# B&R Automation Studio project AS_lab_4
Automation Studio 4.5.2.102

## Configuration Real

### Task classes (Cpu.sw)
```
Cyclic#1 (cycle 2000 us, tolerance 0 us):
  SDCAxisCtr <- SDCAxisCtrlX.prg
  SDCAxisCt1 <- SDCAxisCtrlY.prg
  SDCAxisCt2 <- SDCAxisCtrlZ.prg
DataObjects: Acp10sys
NcDataObjects: acp10etxen <- acp10etxen.dob, Axis_Xa <- AxisParameters.Axis_Xobj.Axis_Xa.dob, Axis_Xi <- AxisParameters.Axis_Xobj.Axis_Xi.dob, gmcipvar <- GmcIpUserConfig.gmcipvar.dob, gmcipfun <- GmcIpUserConfig.gmcipfun.dob, gmcipfub <- GmcIpUserConfig.gmcipfub.dob, gmcipubr <- GmcIpUserConfig.gmcipubr.dob, gmcipusm <- GmcIpUserConfig.gmcipusm.dob, gmcipui <- GmcIpUserConfig.gmcipui.dob, gmcipus <- GmcIpUserConfig.gmcipus.dob, gmcipuc <- GmcIpUserConfig.gmcipuc.dob, gmcipsys <- GmcIpConfig.gmcipsys.dob, gmciplbr <- GmcIpConfig.gmciplbr.dob, gmcipcbr <- GmcIpConfig.gmcipcbr.dob, gmciplsm <- GmcIpConfig.gmciplsm.dob, gmcipcsm <- GmcIpConfig.gmcipcsm.dob, gmcipcfg <- GmcIpConfig.gmcipcfg.dob, gmcipiec <- GmcIpConfig.gmcipiec.dob, gmciplog <- GmcIpConfig.gmciplog.dob, gmcipesm <- GmcIpConfig.gmcipesm.dob, gmcipmxd <- GmcIpConfig.gmcipmxd.dob, gmcipmx <- GmcIpConfig.gmcipmx.dob, CncInit <- CNC.CncInit.dob, CncProg <- CNC.CncProg.dob
VcDataObjects: GUI <- GUI.dob
Binaries: TCData, udbdef, vcpdsw, vcrt, vcmgr, vcctext, vcpfmtcx, vccslider, vcfile, vcgclass, arial, vcdsint, vcdsloc, vcfntttf, GUI01, GUI03, GUI02, vccovl, vcshared, arialbd, vcalarm, vcptelo, vccdt, vcpdpp30, vccbtn, vccnum, vcbclass, vcpfpp30, vctcal, ashwd, Role, User, sysconf, ashwac, asfw, arconfig, iomap, Acp10map, acp10cfg, Acp10map1
Libraries: Acp10man, Acp10par, NcGlobal, Acp10sdc, AsBrStr, Acp10_MC, brsystem, sys_lib, runtime, Acp10sim, AsIOTime, MotorCtrl, powerlnk, vcresman, Arnc0man, DataObj, AsArLog, FileIO, AsArProf, AsMem, astime
```

### Hardware
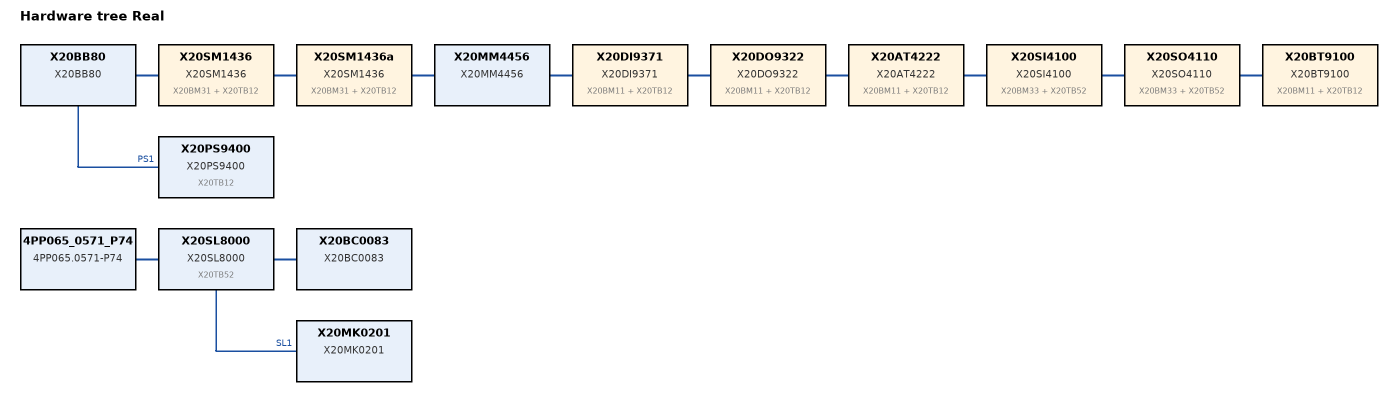
```
4PP065_0571_P74 : 4PP065.0571-P74 v1.1.2.0
  Connector IF5:
    ActivateDevice = 1
    Mode = Manual
    InternetAddress = 10.0.1.10
    SubnetMask = 255.255.255.0
  ConfigurationID = labBR
  Simulation = 1
  TimerDeviceType = EPLX2X
  TimerDevice = 4PP065_0571_P74.IF4
  TaskClassIdleTime = 2000
  Cyclic1Duration = 2000
  Cyclic1Tolerance = 0
  Cyclic1Output = 1
  Cyclic2Duration = 10000
  Cyclic2Tolerance = 10000
  VcObjectName = GUI
X20AT4222 : X20AT4222 v1.2.3.0  [SS1 -> X20TB12e.SS; SL -> X20BM11b.SL1]
X20BB80 : X20BB80 v1.0.2.0
X20BC0083 : X20BC0083 v2.8.0.0  [PLK1 -> X20SL8000.PLK2 [Cable Type=PowerlinkCable, Length=10, Version=1.0.0.2]; SL -> X20BB80.SL1]
X20BM11 : X20BM11 v1.0.0.1  [X2X1 -> X20MM4456.X2X2]
X20BM11a : X20BM11 v1.0.0.1  [X2X1 -> X20BM11.X2X2]
X20BM11b : X20BM11 v1.0.0.1  [X2X1 -> X20BM11a.X2X2]
X20BM11c : X20BM11 v1.0.0.1  [X2X1 -> X20BM33a.X2X2]
X20BM31 : X20BM31 v1.0.0.1  [X2X1 -> X20BB80.IF1]
X20BM31a : X20BM31 v1.0.0.1  [X2X1 -> X20BM31.X2X2]
X20BM33 : X20BM33 v1.0.0.4  [X2X1 -> X20BM11b.X2X2]
X20BM33a : X20BM33 v1.0.0.4  [X2X1 -> X20BM33.X2X2]
X20BT9100 : X20BT9100 v1.0.3.0  [SS1 -> X20TB12f.SS; SL -> X20BM11c.SL1]
X20DI9371 : X20DI9371 v1.0.2.0  [SS1 -> X20TB12c.SS; SL -> X20BM11.SL1]
X20DO9322 : X20DO9322 v1.0.3.0  [SS1 -> X20TB12d.SS; SL -> X20BM11a.SL1]
X20MK0201 : X20MK0201 v1.0.0.0  [SL -> X20SL8000.SL1]
X20MM4456 : X20MM4456 v1.1.5.0  [X2X1 -> X20BM31a.X2X2]
X20PS9400 : X20PS9400 v1.0.2.4  [SS1 -> X20TB12.SS; PS -> X20BB80.PS1]
X20SI4100 : X20SI4100 v1.10.1.1  [SS1 -> X20TB52a.SS; SL -> X20BM33.SL1]
X20SL8000 : X20SL8000 v1.6.5.1  [PLK1 -> 4PP065_0571_P74.IF4 [Cable Type=PowerlinkCable, Length=10, Version=1.0.0.2]; PLK2 -> X20BC0083.PLK1 [Cable Type=PowerlinkCable, Length=10, Version=1.0.0.2]; SS1 -> X20TB52.SS]
  SafeProject = SafeLOGIC-1
X20SM1436 : X20SM1436 v1.4.2.1  [SS1 -> X20TB12a.SS; SL -> X20BM31.SL1]
X20SM1436a : X20SM1436 v1.4.2.1  [SS1 -> X20TB12b.SS; SL -> X20BM31a.SL1]
X20SO4110 : X20SO4110 v1.10.1.1  [SS1 -> X20TB52b.SS; SL -> X20BM33a.SL1]
  SafeModuleID = 3
X20TB12 : X20TB12 v1.0.0.0
X20TB12a : X20TB12 v1.0.0.0
X20TB12b : X20TB12 v1.0.0.0
X20TB12c : X20TB12 v1.0.0.0
X20TB12d : X20TB12 v1.0.0.0
X20TB12e : X20TB12 v1.0.0.0
X20TB12f : X20TB12 v1.0.0.0
X20TB52 : X20TB52 v1.0.0.1
X20TB52a : X20TB52 v1.0.0.1
X20TB52b : X20TB52 v1.0.0.1
```

### IoMap.iom - 4PP065_0571_P74/IoMap.iom
```iecst
VAR_CONFIG
	::PWM_Period AT %QW."X20MM4456".PeriodDurationPWM;
	::SDCAxisCtr:axis_X.PWM AT %QW."X20MM4456".PulseWidthCurrentPWM01;
	::SDCAxisCtr:axis_X.ResetError AT %QX."X20MM4456".ClearError01;
	::SDCAxisCtr:axis_X.ResetCounter AT %QX."X20MM4456".ResetCounter01;
	::SDCAxisCtr:axis_X.Counter AT %IW."X20MM4456".Counter01;
	::SDCAxisCtr:axis_X.EndSwitchA AT %IX."X20MM4456".StatusInput03;
	::SDCAxisCtr:axis_X.EndSwitchB AT %IX."X20MM4456".StatusInput04;
	::SDCAxisCt1:axis_Y.PWM AT %QW."X20MM4456".PulseWidthCurrentPWM02;
	::SDCAxisCt1:axis_Y.ResetError AT %QX."X20MM4456".ClearError02;
	::SDCAxisCt1:axis_Y.ResetCounter AT %QX."X20MM4456".ResetCounter02;
	::SDCAxisCt1:axis_Y.Counter AT %IW."X20MM4456".Counter02;
	::SDCAxisCt1:axis_Y.EndSwitchA AT %IX."X20MM4456".StatusInput07;
	::SDCAxisCt1:axis_Y.EndSwitchB AT %IX."X20MM4456".StatusInput08;
	::SDCAxisCt2:axis_Z.PWM AT %QW."X20MM4456".PulseWidthCurrentPWM03;
	::SDCAxisCt2:axis_Z.ResetCounter AT %QX."X20MM4456".ClearError03;
	::SDCAxisCt2:axis_Z.ResetCounter AT %QX."X20MM4456".ResetCounter03;
	::SDCAxisCt2:axis_Z.Counter AT %IW."X20MM4456".Counter03;
	::SDCAxisCt2:axis_Z.EndSwitchA AT %IX."X20MM4456".StatusInput11;
	::SDCAxisCt2:axis_Z.EndSwitchB AT %IX."X20MM4456".StatusInput12;
	::CoilPWM AT %QW."X20MM4456".PulseWidthCurrentPWM04;
END_VAR
```

### Acp10map1.ncm - 4PP065_0571_P74/Motion/Acp10map1.ncm
```
NcMapping (NcSwId=ACP10, DisabledNodesAreHidden=False)
  NcObject Axis_X (ModuleAddress=SDC_IF1.ST2, InterfaceType=SDC, Type=ncAXIS, Channel=1, AcoposSimulation=Off, InitParameter=Axis_Xi, AcoposParameter=Axis_Xa, AdditionalData=CNC_Enabled="1", Disabled=FALSE, ModuleDisabled=FALSE)
  NcObject Axis_Y (ModuleAddress=SDC_IF1.ST3, InterfaceType=SDC, Type=ncAXIS, Channel=1, AcoposSimulation=Off, InitParameter=Axis_Xi, AcoposParameter=Axis_Xa, AdditionalData=CNC_Enabled="1", Disabled=FALSE, ModuleDisabled=FALSE)
  NcObject Axis_Z (ModuleAddress=SDC_IF1.ST4, InterfaceType=SDC, Type=ncAXIS, Channel=1, AcoposSimulation=Off, InitParameter=Axis_Xi, AcoposParameter=Axis_Xa, AdditionalData=CNC_Enabled="1", Disabled=FALSE, ModuleDisabled=FALSE)
```

### Arnc0cfg.ncc - 4PP065_0571_P74/Motion/Arnc0cfg.ncc
```
NcConfiguration (Version=5.02.1, NcSwId=Arnc0)
  ARNC0CFG_typ:
    sampling_rate = 2000
    cnt_nettrc_rec_drive = 150
    bufsize_sys_trace = 16#00005000
    enable_mp_log = Yes
    tc_nc_man_task = Cyclic #1
    bg_load = 1
    glob_pv_as_ncobject = Yes
```

### Arnc0map.ncm - 4PP065_0571_P74/Motion/Arnc0map.ncm
```
NcMapping (NcSwId=Arnc0, DisabledNodesAreHidden=False)
  NcObject CNCsys (Type=ncCNCSYS, Channel=1, AcoposSimulation=Off, InitParameter=CncInit, Disabled=FALSE, ModuleDisabled=FALSE)
  NcObject CNC24 (Type=ncCNCSYS, Channel=24, AcoposSimulation=Off, Disabled=TRUE, ModuleDisabled=FALSE)
  NcObject CNC23 (Type=ncCNCSYS, Channel=23, AcoposSimulation=Off, Disabled=TRUE, ModuleDisabled=FALSE)
  NcObject CNC22 (Type=ncCNCSYS, Channel=22, AcoposSimulation=Off, Disabled=TRUE, ModuleDisabled=FALSE)
  NcObject CNC21 (Type=ncCNCSYS, Channel=21, AcoposSimulation=Off, Disabled=TRUE, ModuleDisabled=FALSE)
  NcObject CNC20 (Type=ncCNCSYS, Channel=20, AcoposSimulation=Off, Disabled=TRUE, ModuleDisabled=FALSE)
  NcObject CNC19 (Type=ncCNCSYS, Channel=19, AcoposSimulation=Off, Disabled=TRUE, ModuleDisabled=FALSE)
  NcObject CNC18 (Type=ncCNCSYS, Channel=18, AcoposSimulation=Off, Disabled=TRUE, ModuleDisabled=FALSE)
  NcObject CNC17 (Type=ncCNCSYS, Channel=17, AcoposSimulation=Off, Disabled=TRUE, ModuleDisabled=FALSE)
  NcObject CNC16 (Type=ncCNCSYS, Channel=16, AcoposSimulation=Off, Disabled=TRUE, ModuleDisabled=FALSE)
  NcObject CNC15 (Type=ncCNCSYS, Channel=15, AcoposSimulation=Off, Disabled=TRUE, ModuleDisabled=FALSE)
  NcObject CNC14 (Type=ncCNCSYS, Channel=14, AcoposSimulation=Off, Disabled=TRUE, ModuleDisabled=FALSE)
  NcObject CNC13 (Type=ncCNCSYS, Channel=13, AcoposSimulation=Off, Disabled=TRUE, ModuleDisabled=FALSE)
  NcObject CNC12 (Type=ncCNCSYS, Channel=12, AcoposSimulation=Off, Disabled=TRUE, ModuleDisabled=FALSE)
  NcObject CNC11 (Type=ncCNCSYS, Channel=11, AcoposSimulation=Off, Disabled=TRUE, ModuleDisabled=FALSE)
  NcObject CNC10 (Type=ncCNCSYS, Channel=10, AcoposSimulation=Off, Disabled=TRUE, ModuleDisabled=FALSE)
  NcObject CNC9 (Type=ncCNCSYS, Channel=9, AcoposSimulation=Off, Disabled=TRUE, ModuleDisabled=FALSE)
  NcObject CNC8 (Type=ncCNCSYS, Channel=8, AcoposSimulation=Off, Disabled=TRUE, ModuleDisabled=FALSE)
  NcObject CNC7 (Type=ncCNCSYS, Channel=7, AcoposSimulation=Off, Disabled=TRUE, ModuleDisabled=FALSE)
  NcObject CNC6 (Type=ncCNCSYS, Channel=6, AcoposSimulation=Off, Disabled=TRUE, ModuleDisabled=FALSE)
  NcObject CNC5 (Type=ncCNCSYS, Channel=5, AcoposSimulation=Off, Disabled=TRUE, ModuleDisabled=FALSE)
  NcObject CNC4 (Type=ncCNCSYS, Channel=4, AcoposSimulation=Off, Disabled=TRUE, ModuleDisabled=FALSE)
  NcObject CNC3 (Type=ncCNCSYS, Channel=3, AcoposSimulation=Off, Disabled=TRUE, ModuleDisabled=FALSE)
  NcObject CNC2 (Type=ncCNCSYS, Channel=2, AcoposSimulation=Off, Disabled=TRUE, ModuleDisabled=FALSE)
```

## Logical view

Binary libraries used (declarations not repeated): operator, runtime, astime, AsIecCon, Acp10man, Acp10par, NcGlobal, Acp10sdc, AsBrStr, Acp10_MC, brsystem, sys_lib, Acp10sim, AsIOTime, Arnc0man, DataObj, AsArLog, FileIO, AsArProf, AsMem

### Global.var - Global variables
```iecst
VAR
	Axis_X : ACP10AXIS_typ;
	Axis_X_HW : SdcHwCfg_typ;
	Axis_X_EncIf : SdcEncIf16_typ;
	Axis_X_DrvIf : SdcDrvIf16_typ;
	Axis_X_DiDoIf : SdcDiDoIf_typ;
	Axis_Y : ACP10AXIS_typ;
	Axis_Y_HW : SdcHwCfg_typ;
	Axis_Y_EncIf : SdcEncIf16_typ;
	Axis_Y_DrvIf : SdcDrvIf16_typ;
	Axis_Y_DiDoIf : SdcDiDoIf_typ;
	Axis_Z : ACP10AXIS_typ;
	Axis_Z_HW : SdcHwCfg_typ;
	Axis_Z_EncIf : SdcEncIf16_typ;
	Axis_Z_DrvIf : SdcDrvIf16_typ;
	Axis_Z_DiDoIf : SdcDiDoIf_typ;
	PWM_Period : UINT := 200;
	CoilPWM : INT := 0;
	CoilPowered : BOOL;
	CNCsys : ARNC0CNC_typ;
END_VAR
```

### Package Logical/Libraries - Global libraries

### Library Logical/Libraries/MotorCtrl (ANSIC)

#### Types.typ - Exported data types
```iecst
TYPE
	AxisStates :
		(
		STOP := 0,
		HOMING := 1,
		MOVING := 2
		);
END_TYPE
```

#### MotorCtrl.fun - Exported functions and function blocks
```iecst
FUNCTION_BLOCK FB_Regulator
	VAR_INPUT
		e : REAL;
		e_prev : REAL;
	END_VAR
	VAR_OUTPUT
		u : REAL;
	END_VAR
	VAR
		u_raw : REAL;
		k_p : REAL;
		k_i : REAL;
		integrator : FB_Integrator;
		iyOld : REAL;
		max_abs_value : REAL;
	END_VAR
END_FUNCTION_BLOCK

FUNCTION_BLOCK FB_Motor
	VAR_INPUT
		u : REAL;
	END_VAR
	VAR_OUTPUT
		w : REAL;
		phi : REAL;
	END_VAR
	VAR
		integrator : FB_Integrator;
		integrator_phi : FB_Integrator;
		Tm : REAL;
		ke : REAL;
		enable_reg : BOOL;
	END_VAR
END_FUNCTION_BLOCK

FUNCTION_BLOCK FB_Integrator
	VAR_INPUT
		in : REAL;
	END_VAR
	VAR_OUTPUT
		out : REAL;
	END_VAR
	VAR
		dt : REAL;
		direct : BOOL;
	END_VAR
END_FUNCTION_BLOCK

FUNCTION_BLOCK FB_Axis
	VAR_INPUT
		U : REAL;
		UserSpeed : INT;
		EndSwitchA : BOOL;
		EndSwitchB : BOOL;
		ForceSwitchA : BOOL;
		ForceSwitchB : BOOL;
		Counter : INT;
		UserResetCounter : BOOL;
	END_VAR
	VAR_OUTPUT
		FeedbackSpeed : REAL;
		PWM : INT;
		ResetError : BOOL;
		ResetCounter : BOOL;
	END_VAR
	VAR
		MaxSpeed : UINT;
		Manual : BOOL;
	END_VAR
END_FUNCTION_BLOCK
```

#### FB_Regulator.c
```c
#include <bur/plctypes.h>
#ifdef __cplusplus
	extern "C"
	{
#endif
#include "MotorCtrl.h"
#ifdef __cplusplus
	};
#endif

#include "Math.h"
/* TODO: Add your comment here */
void FB_Regulator(struct FB_Regulator* inst)
{
	if (inst->integrator.direct)
		inst->integrator.in = inst->k_i * inst->e_prev + inst->iyOld / inst->integrator.dt;
	else
		inst->integrator.in = inst->k_i * inst->e + inst->iyOld / inst->integrator.dt;
	FB_Integrator(&inst->integrator);
	inst->u_raw = (fabs(inst->k_p * inst->e) < inst->max_abs_value ? inst->k_p * inst->e : inst->max_abs_value * copysign(1.0, inst->k_p * inst->e)) + inst->integrator.out;
	inst->u = fabs(inst->u_raw) < inst->max_abs_value ? inst->u_raw : inst->max_abs_value * copysign(1.0, inst->u_raw);
	inst->iyOld = inst->u - inst->u_raw;
}
```

#### FB_Axis.c
```c
#include <bur/plctypes.h>
#ifdef __cplusplus
	extern "C"
	{
#endif
#include "MotorCtrl.h"
#ifdef __cplusplus
	};
#endif

#include "math.h"
/* TODO: Add your comment here */
void FB_Axis(struct FB_Axis* inst)
{
	inst->ResetError = inst->ResetCounter = 0;

	if (inst->UserResetCounter)
	{
		inst->ResetCounter = 1;
		inst->UserResetCounter = 0;
	}

	inst->PWM = (int)round(inst->U / 24.0 * 32767.0);
	inst->FeedbackSpeed = inst->U / 24.0 * inst->MaxSpeed;

	if (inst->EndSwitchA || inst->EndSwitchB)
	{
		inst->ResetError = 1;
		inst->PWM = 0;
	}
}
```

### Program Logical/SDCAxisCtrlX (ANSIC)

#### Variables.var
```iecst
VAR
	axis_X : FB_Axis;
	Regulator : FB_Regulator;
END_VAR
```

#### Main.c
```c
#include <bur/plctypes.h>

#ifdef _DEFAULT_INCLUDES
#include <AsDefault.h>
#endif

void _INIT ProgramInit(void)
{
	//Устанавливаем типы SDC модулей
	Axis_X_HW.EncIf1_Typ = ncSDC_ENC16;
	Axis_X_HW.DiDoIf_Typ = ncSDC_DIDO;
	Axis_X_HW.DrvIf_Typ = ncSDC_DRVSERVO16;

	//Устанавливаем имена переменных
	strcpy(Axis_X_HW.EncIf1_Name, "Axis_X_EncIf");
	strcpy(Axis_X_HW.DrvIf_Name, "Axis_X_DrvIf");
	strcpy(Axis_X_HW.DiDoIf_Name, "Axis_X_DiDoIf");

	//Устанавливаем входы готовности и нормальной работы
	Axis_X_EncIf.iEncOK = 1;
	Axis_X_DrvIf.iDrvOK = 1;
	Axis_X_DrvIf.iStatusEnable = 1;
	Axis_X_DiDoIf.iDriveReady = 1;

	Regulator.integrator.dt = 0.002;
	Regulator.integrator.direct = 0;
	Regulator.k_i = 0.16;
	Regulator.k_p = 0.0001;
	Regulator.max_abs_value = 24.0;

	axis_X.MaxSpeed = 6500;
}

void _CYCLIC ProgramCyclic(void)
{
	Axis_X_EncIf.iLifeCnt++;
	Axis_X_DiDoIf.iLifeCntDriveEnable++;
	Axis_X_DiDoIf.iLifeCntDriveReady++;
	Axis_X_DiDoIf.iLifeCntNegHwEnd++;
	Axis_X_DiDoIf.iLifeCntPosHwEnd++;
	Axis_X_DiDoIf.iLifeCntReference++;
	Axis_X_DrvIf.iLifeCnt++;

	Axis_X_EncIf.iActTime = (INT)	AsIOTimeCyclicStart();
	Axis_X_EncIf.iActPos = axis_X.Counter;

	Axis_X_DiDoIf.iPosHwEnd = (axis_X.EndSwitchA || axis_X.ForceSwitchA);
	Axis_X_DiDoIf.iNegHwEnd = (axis_X.EndSwitchB || axis_X.ForceSwitchB);

	CoilPWM = CoilPowered ? 32767 : 0;

	if (CoilPowered)
	{
		Regulator.e = (axis_X.Manual ? axis_X.UserSpeed : Axis_X_DrvIf.oSetPos * 6500.0 / 32767.0) - axis_X.FeedbackSpeed;
		FB_Regulator(&Regulator);

		axis_X.U = Regulator.u;
		FB_Axis(&axis_X);
	}
	else
	{
		axis_X.PWM = 0;
	}
}

void _EXIT ProgramExit(void)
{
	// Insert code here

}
```

### Program Logical/SDCAxisCtrlY (ANSIC)

#### Variables.var
```iecst
VAR
	axis_Y : FB_Axis;
	Regulator : FB_Regulator;
END_VAR
```

#### Main.c
```c
#include <bur/plctypes.h>

#ifdef _DEFAULT_INCLUDES
#include <AsDefault.h>
#endif

void _INIT ProgramInit(void)
{
	//Устанавливаем типы SDC модулей
	Axis_Y_HW.EncIf1_Typ = ncSDC_ENC16;
	Axis_Y_HW.DiDoIf_Typ = ncSDC_DIDO;
	Axis_Y_HW.DrvIf_Typ = ncSDC_DRVSERVO16;

	//Устанавливаем имена переменных
	strcpy(Axis_Y_HW.EncIf1_Name, "Axis_Y_EncIf");
	strcpy(Axis_Y_HW.DrvIf_Name, "Axis_Y_DrvIf");
	strcpy(Axis_Y_HW.DiDoIf_Name, "Axis_Y_DiDoIf");

	//Устанавливаем входы готовности и нормальной работы
	Axis_Y_EncIf.iEncOK = 1;
	Axis_Y_DrvIf.iDrvOK = 1;
	Axis_Y_DrvIf.iStatusEnable = 1;
	Axis_Y_DiDoIf.iDriveReady = 1;

	Regulator.integrator.dt = 0.002;
	Regulator.integrator.direct = 0;
	Regulator.k_i = 0.16;
	Regulator.k_p = 0.0001;
	Regulator.max_abs_value = 24.0;

	axis_Y.MaxSpeed = 6500;
}

void _CYCLIC ProgramCyclic(void)
{
	Axis_Y_EncIf.iLifeCnt++;
	Axis_Y_DiDoIf.iLifeCntDriveEnable++;
	Axis_Y_DiDoIf.iLifeCntDriveReady++;
	Axis_Y_DiDoIf.iLifeCntNegHwEnd++;
	Axis_Y_DiDoIf.iLifeCntPosHwEnd++;
	Axis_Y_DiDoIf.iLifeCntReference++;
	Axis_Y_DrvIf.iLifeCnt++;

	Axis_Y_EncIf.iActTime = (INT)	AsIOTimeCyclicStart();
	Axis_Y_EncIf.iActPos = axis_Y.Counter;

	Axis_Y_DiDoIf.iPosHwEnd = (axis_Y.EndSwitchA || axis_Y.ForceSwitchA);
	Axis_Y_DiDoIf.iNegHwEnd = (axis_Y.EndSwitchB || axis_Y.ForceSwitchB);

	CoilPWM = CoilPowered ? 32767 : 0;

	if (CoilPowered)
	{
		Regulator.e = (axis_Y.Manual ? axis_Y.UserSpeed : Axis_Y_DrvIf.oSetPos * 6500.0 / 32767.0) - axis_Y.FeedbackSpeed;
		FB_Regulator(&Regulator);

		axis_Y.U = Regulator.u;
		FB_Axis(&axis_Y);
	}
	else
	{
		axis_Y.PWM = 0;
	}
}

void _EXIT ProgramExit(void)
{
	// Insert code here

}
```

### Program Logical/SDCAxisCtrlZ (ANSIC)

#### Variables.var
```iecst
VAR
	axis_Z : FB_Axis;
	Regulator : FB_Regulator;
END_VAR
```

#### Main.c
```c
#include <bur/plctypes.h>

#ifdef _DEFAULT_INCLUDES
#include <AsDefault.h>
#endif

void _INIT ProgramInit(void)
{
	//Устанавливаем типы SDC модулей
	Axis_Z_HW.EncIf1_Typ = ncSDC_ENC16;
	Axis_Z_HW.DiDoIf_Typ = ncSDC_DIDO;
	Axis_Z_HW.DrvIf_Typ = ncSDC_DRVSERVO16;

	//Устанавливаем имена переменных
	strcpy(Axis_Z_HW.EncIf1_Name, "Axis_Z_EncIf");
	strcpy(Axis_Z_HW.DrvIf_Name, "Axis_Z_DrvIf");
	strcpy(Axis_Z_HW.DiDoIf_Name, "Axis_Z_DiDoIf");

	//Устанавливаем входы готовности и нормальной работы
	Axis_Z_EncIf.iEncOK = 1;
	Axis_Z_DrvIf.iDrvOK = 1;
	Axis_Z_DrvIf.iStatusEnable = 1;
	Axis_Z_DiDoIf.iDriveReady = 1;

	Regulator.integrator.dt = 0.002;
	Regulator.integrator.direct = 0;
	Regulator.k_i = 0.16;
	Regulator.k_p = 0.0001;
	Regulator.max_abs_value = 24.0;

	axis_Z.MaxSpeed = 6500;
}

void _CYCLIC ProgramCyclic(void)
{
	Axis_Z_EncIf.iLifeCnt++;
	Axis_Z_DiDoIf.iLifeCntDriveEnable++;
	Axis_Z_DiDoIf.iLifeCntDriveReady++;
	Axis_Z_DiDoIf.iLifeCntNegHwEnd++;
	Axis_Z_DiDoIf.iLifeCntPosHwEnd++;
	Axis_Z_DiDoIf.iLifeCntReference++;
	Axis_Z_DrvIf.iLifeCnt++;

	Axis_Z_EncIf.iActTime = (INT)	AsIOTimeCyclicStart();
	Axis_Z_EncIf.iActPos = axis_Z.Counter;

	Axis_Z_DiDoIf.iPosHwEnd = (axis_Z.EndSwitchA || axis_Z.ForceSwitchA);
	Axis_Z_DiDoIf.iNegHwEnd = (axis_Z.EndSwitchB || axis_Z.ForceSwitchB);

	CoilPWM = CoilPowered ? 32767 : 0;

	if (CoilPowered)
	{
		Regulator.e = (axis_Z.Manual ? axis_Z.UserSpeed : Axis_Z_DrvIf.oSetPos * 6500.0 / 32767.0) - axis_Z.FeedbackSpeed;
		FB_Regulator(&Regulator);

		axis_Z.U = Regulator.u;
		FB_Axis(&axis_Z);
	}
	else
	{
		axis_Z.PWM = 0;
	}
}

void _EXIT ProgramExit(void)
{
	// Insert code here

}
```

### Package Logical/AxisParameters/Axis_Xobj - Axis_Xobj

### Data object Logical/AxisParameters/Axis_Xobj/Axis_Xi (Ax)

#### Axis_Xi.ax - ACP10 init object for axis
```
InitParameter (Version=5.2.1, NcSwId=ACP10)
  ACP10AXIS_typ:
    dig_in:
      level:
        reference = ncACTIV_HI
        pos_hw_end = ncACTIV_HI
        neg_hw_end = ncACTIV_HI
        trigger1 = ncACTIV_HI
        trigger2 = ncACTIV_HI
    encoder_if:
      parameter:
        count_dir = ncSTANDARD
        scaling:
          load:
            units = 3000
            rev_motor = 1
    limit:
      parameter:
        v_pos = 10000.0
        v_neg = 10000.0
        a1_pos = 10000.0
        a2_pos = 10000.0
        a1_neg = 10000.0
        a2_neg = 10000.0
        t_jolt = 0.0
        t_in_pos = 0.0
        pos_sw_end = 8388607
        neg_sw_end = -8388608
        ds_warning = 500.0
        ds_stop = 50000.0
        a_stop = 1.0E+30
        dv_stop = 0.0
        dv_stop_mode = ncOFF
    controller:
      mode = ncPOSITION
      position:
        kv = 10.0
        tn = 0.0
        t_predict = 0.0004
        t_total = 0.0004
        p_max = 1.0E+30
        i_max = 0.0
      speed:
        kv = 2.0
        tn = 0.0
        t_filter = 0.0
        isq_filter1:
          type = ncOFF
          a0 = 0.0
          a1 = 0.0
          b0 = 0.0
          b1 = 0.0
          b2 = 0.0
          c0_par_id = 0
          c1_par_id = 0
        isq_filter2:
          type = ncOFF
          a0 = 0.0
          a1 = 0.0
          b0 = 0.0
          b1 = 0.0
          b2 = 0.0
          c0_par_id = 0
          c1_par_id = 0
        isq_filter3:
          type = ncOFF
          a0 = 0.0
          a1 = 0.0
          b0 = 0.0
          b1 = 0.0
          b2 = 0.0
          c0_par_id = 0
          c1_par_id = 0
      uf:
        type = ncLINEAR + ncCORRECTION
        auto_config = ncMOTOR_PAR
        u0 = 0.0
        un = 0.0
        fn = 50.0
        k_f_slip = 0.0
      ff:
        torque_load = 0.0
        torque_pos = 0.0
        torque_neg = 0.0
        kv_torque = 0.0
        inertia = 0.0
        t_filter_a = 0.0
    move:
      stop:
        parameter[0]:
          decel_ramp = ncA_LIMIT
          controller = ncON
        parameter[1]:
          decel_ramp = ncA_LIMIT
          controller = ncON
        parameter[2]:
          decel_ramp = ncA_LIMIT
          controller = ncON
        parameter[3]:
          decel_ramp = ncA_LIMIT
          controller = ncON
        quickstop:
          decel_ramp = ncA_LIMIT
          t_jolt = 0.0
        drive_error:
          decel_ramp = ncA_LIMIT
      homing:
        parameter:
          s = 0
          v_switch = 6000.0
          v_trigger = 2000.0
          a = 10000.0
          mode = ncDIRECT
          edge_sw = ncNEGATIVE
          start_dir = ncPOSITIVE
          trigg_dir = ncNEGATIVE
          ref_pulse = ncOFF
          fix_dir = ncOFF
          tr_s_block = 0.0
          torque_lim = 0.0
          ds_block = 0.0
          ds_stop = 0.0
      basis:
        parameter:
          v_pos = 5000.0
          v_neg = 5000.0
          a1_pos = 10000.0
          a2_pos = 10000.0
          a1_neg = 10000.0
          a2_neg = 10000.0
    message:
      text:
        parameter:
          format = ncBREAK
          columns = 80
          data_modul = acp10etxen
```

- Visualisation Logical/GUI (not shown)

### Data object Logical/CncInit (Cns)

- CncInit.cns (not shown)

### Data object Logical/CncProg (Cnc)

#### CncProg.cnc
```
(AxisLength: 36 cm, 2000 units)
(Translation: 2000 / 36 * 10 = 555.56 real-units)
(DriveSpeed: 24 * 145 / 60 = 58 real-units/s)
(AxisSpeed: 6500 virtual-units/s)
(Hence, Translation [virtual-units] = AxisSpeed / DriveSpeed * Translation [real-units] = )
( = 6500 / 58 * 555.56 = 62260 virtual-units)

%001 (CncProgram)
N05 G90
N10 F390000
N20 G01 X0 Y62260 Z0
N30 G01 X0 Y62260 Z62260
N40 G01 X62260 Y0 Z62260
N50 G01 X0 Y0 Z62260
N60 G01 X0 Y0 Z0
N999 M30
```

Listed in the project but not available here: Logical/Global.typ, Logical/Libraries/MotorCtrl/Constants.var, Logical/Libraries/MotorCtrl/FB_Motor.c, Logical/Libraries/MotorCtrl/FB_Integrator.c, Logical/acp10etxen, Logical/GmcIpConfig, Logical/GmcIpUserConfig
